// TIA Portal V16 export
// export: Created 2024-04-26T21:24:42.9249346Z, ExportSetting WithDefaults, DisplayName Totally Integrated Automation Portal, DisplayVersion V16, DisplayName TIA Portal Version Control Interface, DisplayVersion V16, DisplayName TIA Portal Openness, DisplayVersion V16, DisplayName STEP 7 Professional, DisplayVersion V16, DisplayName STEP 7 Safety, DisplayVersion V16, DisplayName WinCC Professional, DisplayVersion V16
DATA_BLOCK "MC_Reset_DB_1"   // DB13
// stored: AutoNumber true, InstanceOfName MC_Reset, OfSystemLibElement MC_Reset, OfSystemLibVersion 6.0
"MC_Reset"
   // VAR_INPUT
   //    Axis : TO_Axis;
   //    Execute : Bool;
   //    Restart : Bool;
   // END_VAR
   // VAR_OUTPUT
   //    Done : Bool;
   //    Busy : Bool;
   //    Error : Bool;
   //    ErrorID : Word;
   //    ErrorInfo : Word;
   // END_VAR
   // VAR
   //    FB_ID : DInt;
   // END_VAR
BEGIN
END_DATA_BLOCK
